FUNCTION_BLOCK Actuator_Fault_CAT_HMI (* Service Interface Function Block Type *)
  (* Standard: 61499-2 *)
  (* Version 0.0, 2/24/2026, Schneider Electric, template *)
  PACKAGE Main;
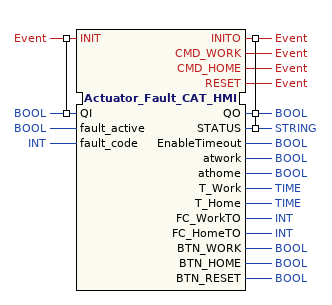
  EVENT_INPUT
    INIT WITH QI;
  END_EVENT
  EVENT_OUTPUT
    INITO WITH QO, STATUS;
    CMD_WORK;
    CMD_HOME;
    RESET;
  END_EVENT
  VAR_INPUT
    QI : BOOL;
    fault_active : BOOL;
    fault_code : INT;
  END_VAR
  VAR_OUTPUT
    QO : BOOL; (* Event Output Qualifier *)
    STATUS : STRING; (* Service Status *)
    EnableTimeout : BOOL;
    atwork : BOOL;
    athome : BOOL;
    T_Work : TIME;
    T_Home : TIME;
    FC_WorkTO : INT;
    FC_HomeTO : INT;
    BTN_WORK : BOOL;
    BTN_HOME : BOOL;
    BTN_RESET : BOOL;
  END_VAR
  SERVICE /
    SEQUENCE 
    END_SEQUENCE
  END_SERVICE
END_FUNCTION_BLOCK
